TYPE T_PackMLMode : UINT;
END_TYPE

(* stored: Version 1.1.0.1, ProductVersion 3.1.4026.18
   DUT T_PackMLMode: Id {5fd115b1-902a-420b-bf04-3e5e78af9a90} *)
